FUNCTION_BLOCK RecordStartTime
VAR_INPUT
	StartFlag: BOOL := FALSE;
END_VAR
VAR_OUTPUT
	RecordStFinish : BOOL :=FALSE;
	BeginLo: UDINT;
	BeginHi: UDINT;
END_VAR
VAR
	UpTrigDetect: R_TRIG;
	MyTimer: getsystemtime;
	Delay: TON;
END_VAR

//start to get system time
MyTimer();

//detect the trigger: false to true
UpTrigDetect(CLK:=StartFlag);

//record beginning Timestamp of initializing period
IF UpTrigDetect.Q THEN
	BeginLo := MyTimer.timeLoDW;								
	BeginHi := MyTimer.timeHiDW;
END_IF

RecordStFinish := TRUE;

END_FUNCTION_BLOCK

(* stored: Version 1.1.0.1, ProductVersion 3.1.4024.3
   POU RecordStartTime: Id {97d78cee-8bd9-496e-8a02-6d3fa1e4fe07}, SpecialFunc None *)
